{attribute 'linkalways'} 
{attribute 'no_explicit_call' := 'This FB is a CLASS and must be accessed using methods or properties'}
{attribute 'enable_dynamic_creation'}
FUNCTION_BLOCK _SINT EXTENDS NumericDatatypeBase
VAR
	localData : SINT;
	activeData : REFERENCE TO SINT REF= localData;
END_VAR

PROPERTY PUBLIC Address : PVOID
GET
Address := ADR(activeData);
END_GET
END_PROPERTY

METHOD PUBLIC ClearReference
VAR_INPUT
END_VAR
activeData REF= localData;
END_METHOD

METHOD PUBLIC Clone : I_Datatype
VAR
    pClone : POINTER TO _SINT;
END_VAR
pClone := __NEW(_SINT(InitialValue := Value));
Clone := pClone^;
END_METHOD

METHOD FB_init : BOOL
VAR_INPUT
	bInitRetains : BOOL; // if TRUE, the retain variables are initialized (warm start / cold start)
	bInCopyCode : BOOL;  // if TRUE, the instance afterwards gets moved into the copy code (online change)
	InitialValue : SINT;
END_VAR
localData := InitialValue;
END_METHOD

PROPERTY PUBLIC IsFloat : BOOL
GET
IsFloat := FALSE;
END_GET
END_PROPERTY

PROPERTY PUBLIC IsSigned : BOOL
GET
IsSigned := TRUE;
END_GET
END_PROPERTY

METHOD PUBLIC MakeReferenceTo
VAR_INPUT
	ReferenceTarget : REFERENCE TO SINT;
END_VAR
activeData REF= ReferenceTarget;
END_METHOD

PROPERTY PUBLIC MaxValue : SINT
GET
MaxValue :=  DatatypeLimits.SINT_MAX_VALUE;
END_GET
END_PROPERTY

PROPERTY PUBLIC MinValue : SINT
GET
MinValue := DatatypeLimits.SINT_MIN_VALUE;
END_GET
END_PROPERTY

METHOD PROTECTED SerializeMaxValue
VAR_INPUT
	Serializer : I_Serializer;
END_VAR
Serializer.AddSint(MaxValue);
END_METHOD

METHOD PROTECTED SerializeMinValue
VAR_INPUT
	Serializer : I_Serializer;
END_VAR
Serializer.AddSint(MinValue);
END_METHOD

METHOD PUBLIC SerializeWith
VAR_INPUT
	Serializer : I_Serializer;
END_VAR
Serializer.AddSint(activeData);
END_METHOD

PROPERTY PUBLIC Size : UDINT
GET
Size := SIZEOF(activeData);
END_GET
END_PROPERTY

METHOD TryDeserializeFrom : BOOL
VAR_INPUT
	Deserializer : I_Deserializer;
	Feedback : I_DeserializerFeedback;
END_VAR
TryDeserializeFrom := Deserializer.TryGetSint(activeData, Feedback);
END_METHOD

METHOD TryMakeReferenceTo : BOOL
VAR_INPUT
	Target : I_Datatype;
END_VAR
VAR
	pTargetData : POINTER TO SINT;
END_VAR
IF NOT (Target.TypeName = TypeName) THEN
	RETURN;
END_IF

pTargetData := Target.Address;
activeData REF= pTargetData^;
TryMakeReferenceTo := TRUE;
END_METHOD

PROPERTY PUBLIC TypeName : T_MAXSTRING
GET
TypeName := 'SINT';
END_GET
END_PROPERTY

PROPERTY PUBLIC Value : REFERENCE TO SINT
GET
Value REF= activeData;
END_GET
END_PROPERTY

END_FUNCTION_BLOCK

(* stored: Version 1.1.0.1, ProductVersion 3.1.4024.12
   POU _SINT: Id {baa9b623-38b4-4986-b596-0141fbde1188}, SpecialFunc None
   Folder Constructor: Id {ca89985d-f8c7-40b2-a1d5-e0d5851c326e}
   Folder Protected: Id {e1688de6-9cb9-4e39-874d-681a2ea0cdf2}
   Property Address: Id {e5591d7a-20a4-47b5-9b6a-cd3d6df4a536}
   Get Get: Id {3e338be3-098a-499b-99e4-7d5654b4df55}
   Method ClearReference: Id {75f32e98-47a8-4b25-b8ce-365065b3dd76}
   Method Clone: Id {d8cdc587-602c-4f46-aae6-733fe2135ead}
   Method FB_init: Id {4f2eaad4-b352-4e27-a9f9-ca3e9cf75256}
   Property IsFloat: Id {8de4cb73-0e9a-4aa4-8ec8-40c4688ae390}
   Get Get: Id {7a810fa6-bc0a-4893-8914-1be8ec9e8498}
   Property IsSigned: Id {dafa3d29-c8e7-40b7-a122-2cdeaa862b48}
   Get Get: Id {e116f197-2b4d-4f57-aad1-644d3835c8df}
   Method MakeReferenceTo: Id {a920b83e-637d-46e7-85b7-92b694f42757}
   Property MaxValue: Id {be11f9d7-6c2b-4c49-bf0e-7c9accea8d8a}
   Get Get: Id {fa5f5f1b-f2c8-4088-b33c-588aa85a067a}
   Property MinValue: Id {cd63a22a-47f3-4138-98f7-342494154acf}
   Get Get: Id {82966c25-6ebf-439f-ae8b-7f2f1aab64a7}
   Method SerializeMaxValue: Id {667af442-38a6-463f-82ae-0ef3929094c3}
   Method SerializeMinValue: Id {858ea518-cf2a-416b-a1cf-b4ed46a6198f}
   Method SerializeWith: Id {c03e7885-a45b-454a-b086-a264e38aba89}
   Property Size: Id {7e65ccc3-fb06-441d-9dbe-d0120a34c432}
   Get Get: Id {1065f0ec-754b-492b-9e7e-7df73c1b3900}
   Method TryDeserializeFrom: Id {f4559769-7aee-4116-8595-a5c4be5f1abf}
   Method TryMakeReferenceTo: Id {6b72bdcb-b9c0-4ff0-a0a2-e2658d3c6d80}
   Property TypeName: Id {660c5a4e-0377-4c67-b8ff-c621785afcaa}
   Get Get: Id {02178733-005a-4eff-a41e-e00687adebb2}
   Property Value: Id {12f26868-cd97-476b-9f8a-949fc5908bbf}
   Get Get: Id {2aa5fc95-a94b-4cd0-b411-6160dabbae69} *)
